ABB RobotStudio station: Lab_robotica_g6.rsstn

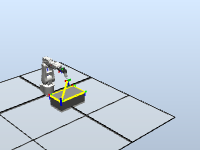
Station Solution97 (saved by RobotStudio 6.6.7701.1025)
Controller IRB_120_3kg_0.58m
  mechanical unit ROB_1: IRB120_3_58__01, 6 joints, base frame (0, 0, 0) mm
Layout (positions relative to the parent item):
  - IRB120_3_58__01 [mechanism, from Robots\IRB120_3_58_G_01.rslib] at (0, 0, 0) mm; joint values [0, 0, 0, 0, 0.5236, 0] (rad or m)
  - MyTool [mechanism, from Training Objects\myTool.rslib] at (364.35, 0, 594) mm, rotated rx 180 ry 60 rz 180 deg
  - Pieza_5 [part] at (624.59, -204.58, -30.2) mm, rotated rx 0 ry 0 rz 90 deg
Attachment: MyTool is attached to IRB120_3_58__01 / Link6
Attachment: Workobject_caja is attached to Pieza_5
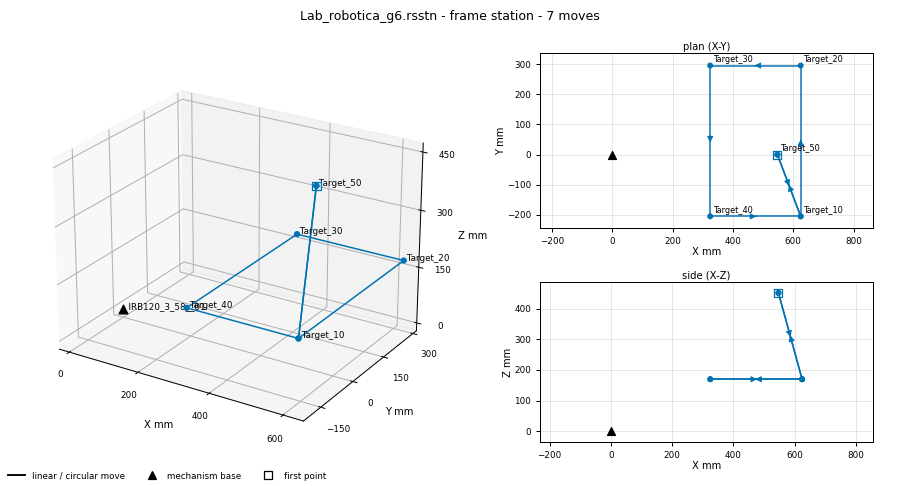
[picture p0: tool path of Lab_robotica_g6.rsstn in frame station, 7 of 7 moves have a stored position in this frame; points joined in program order, loops and branches not executed]
Targets, tools, work objects and paths stored in the station, written as RAPID:
! task (no controller)
MODULE Module1
  CONST robtarget Target_50:=[[99.315262647,380.36695645,-251.647267557],[0.694115243,-0.134922307,-0.134922307,-0.694115243],[0,0,0,0],[9E+09,9E+09,9E+09,9E+09,9E+09,9E+09]];
ENDMODULE

! task T_ROB1
MODULE CalibData
  PERS tooldata MyTool:=[TRUE,[[31.792631019,0,229.638935148],[0.945518576,0,0.325568154,0]],[1,[0,0,1],[1,0,0,0],0,0,0]];
  TASK PERS wobjdata Workobject_caja:=[FALSE,TRUE,"",[[624.592699382,-204.583259915,169.803210722],[0.707106781,0,0,0.707106781]],[[0,0,0],[0,0.707106781,0.707106781,0]]];
ENDMODULE

! task T_ROB1
MODULE Module1
  CONST robtarget Target_10:=[[0,0,0],[1,0,0,0],[0,0,0,0],[9E+09,9E+09,9E+09,9E+09,9E+09,9E+09]];
  CONST robtarget Target_20:=[[0,500,0],[1,0,0,0],[0,0,0,0],[9E+09,9E+09,9E+09,9E+09,9E+09,9E+09]];
  CONST robtarget Target_30:=[[300,500,0],[1,0,0,0],[0,0,0,0],[9E+09,9E+09,9E+09,9E+09,9E+09,9E+09]];
  CONST robtarget Target_40:=[[300,0,0],[1,0,0,0],[0,0,0,0],[9E+09,9E+09,9E+09,9E+09,9E+09,9E+09]];
  CONST robtarget Target_50:=[[547.330680325,0,451.647267557],[0.190808957,0,0.981627191,0],[0,0,0,0],[9E+09,9E+09,9E+09,9E+09,9E+09,9E+09]];
  PROC Path_10()
    MoveL Target_50,v100,fine,MyTool\WObj:=wobj0;
    MoveL Target_10,v100,fine,MyTool\WObj:=Workobject_caja;
    MoveL Target_20,v100,fine,MyTool\WObj:=Workobject_caja;
    MoveL Target_30,v100,fine,MyTool\WObj:=Workobject_caja;
    MoveL Target_40,v100,fine,MyTool\WObj:=Workobject_caja;
    MoveL Target_10,v100,fine,MyTool\WObj:=Workobject_caja;
    MoveL Target_50,v100,fine,MyTool\WObj:=wobj0;
  ENDPROC
ENDMODULE

